# EPICS substitutions: mc14/db/pmac_asyn_motor.substitutions
file "db/pmac_asyn_motor.db"
{
pattern
{SYS,            DEV,                   MOTOR,  SPORT,  ADDR,  DESC,       DTYP        PREC,  EGU }
{"XF:23ID2-ES",  "{APPES:1-Ax:X}",  "M0",   "P0",  1,     "APPES X",    asynMotor,  3,     "mm"  }
{"XF:23ID2-ES",  "{APPES:1-Ax:Y}",  "M0",   "P0",  2,     "APPES Y",    asynMotor,  3,     "mm"  }
{"XF:23ID2-ES",  "{APPES:1-Ax:Z}",  "M0",   "P0",  3,     "APPES Z",    asynMotor,  3,     "mm"  }
{"XF:23ID2-ES",  "{APPES:1-Ax:R}",  "M0",   "P0",  4,     "APPES R",    asynMotor,  3,     "mm"  }
}
